FUNCTION_BLOCK T_RoboConnect_SetToolDigitalOutputTimeout_Fails EXTENDS T_UnitTestBase
VAR
  robot : I_RoboConnect;
  timeOutTimer : TON;
  targetDO : UINT;
  myTestState, prevState :
    (INIT, ARRANGE, ACT, ASSERT) := INIT;
  expected, actual : BOOL;
  counter : UINT;
END_VAR

CASE myTestState OF
  INIT:
    StateChanged();
    myTestState := ARRANGE;

  ARRANGE:
    IF StateChanged() THEN
      expected := TRUE;
      robot.Connect();
    END_IF

    IF robot.Connected THEN
      myTestState := ACT;
    END_IF

  ACT:
    robot.SetToolDigitalOutput(targetDO,TRUE);
    myTestState := ASSERT;

  ASSERT:

    IF timeOutTimer.Q THEN
      actual := robot.GetToolDigitalOutput(targetDO);
      assertion.AssertEquals_BOOL(expected, actual, 'robot.GetDigitalOutput(targetDO) := TRUE');
      TestFinished();
      myTestState := INIT;

    END_IF

END_CASE

timeOutTimer(IN := myTestState = ASSERT);

METHOD FB_init : BOOL
VAR_INPUT
  bInitRetains : BOOL; // if TRUE, the retain variables are initialized (warm start / cold start)
  bInCopyCode : BOOL; // if TRUE, the instance afterwards gets moved into the copy code (online change)
  TestSuite : tcl_SimpleUnitTestLibrary.I_TestSuite;
  robot : I_TcRobot;
  timeout : TIME;
  targetDo : UINT;
END_VAR
THIS^.robot := robot;
THIS^.timeOutTimer.PT := timeout;
THIS^.targetDo := targetDo;
END_METHOD

METHOD PRIVATE StateChanged : BOOL
IF  myTestState = prevState THEN
  RETURN;
END_IF

prevState := myTestState;
StateChanged := TRUE;
END_METHOD

METHOD WaitForCycles : BOOL
VAR_INPUT
  maxCount : UINT;
END_VAR
counter := counter + 1;

IF counter = maxCount THEN
  counter := 0;
  WaitForCycles := TRUE;
END_IF
END_METHOD

END_FUNCTION_BLOCK

(* stored: Version 1.1.0.1
   POU T_TcRobot_SetToolDigitalOutputTimeout_Fails: Id {a7736064-db0e-4ad2-8d4b-8e2cdf85128d}, SpecialFunc None
   Method FB_init: Id {af461771-3c8a-4957-b195-071ad06f71c8}
   Method StateChanged: Id {6a4ada68-633b-4b64-b8a2-c220b731c8c4}
   Method WaitForCycles: Id {3babe237-5e24-4731-a60a-6ef4cc2dcda3} *)
